TYPE (* logiBUS AI Struct Octal *)
  (* Version 1.0, 2026-05-28, franz *)
  PACKAGE logiBUS::io::AI;
  IMPORT eclipse4diac::core::TypeHash;
  IMPORT logiBUS::io::AI::logiBUS_AI_S;
  logiBUS_AI_S_Octal : STRUCT
    Port1 : logiBUS_AI_S := (Pin := 255);
    Port2 : logiBUS_AI_S := (Pin := 255);
    Port3 : logiBUS_AI_S := (Pin := 255);
    Port4 : logiBUS_AI_S := (Pin := 255);
    Port5 : logiBUS_AI_S := (Pin := 255);
    Port6 : logiBUS_AI_S := (Pin := 255);
    Port7 : logiBUS_AI_S := (Pin := 255);
    Port8 : logiBUS_AI_S := (Pin := 255);
  END_STRUCT;
END_TYPE
